(* IEC 61131-3 sources: Conveyor/test/Mocks, 7 files *)

(* ---- MockingAutoRelease copy.st ---- *)
USING Simatic.Ax.IO.Input;
NAMESPACE Simatic.Ax.Conveyor.Mocks

    CLASS MockBinSignal
        IMPLEMENTS IBinSignal
        VAR PUBLIC
            QValue : BOOL;
            QRisValue : BOOL;
            QFalValue : BOOL;
        END_VAR

        METHOD PUBLIC Q : BOOL
            Q := QValue;
        END_METHOD

        METHOD PUBLIC QRis : BOOL
            QRis := QRisValue;
        END_METHOD

        METHOD PUBLIC QFal : BOOL
            QFal := QFalValue;
        END_METHOD

        METHOD PUBLIC QBad : BOOL
            ;
        END_METHOD
END_CLASS
END_NAMESPACE

(* ---- MockingAutoRelease.st ---- *)
USING Simatic.Ax.AutomationBase;
NAMESPACE Simatic.Ax.Conveyor.Mocks

    CLASS MockAutoStartup
        IMPLEMENTS IAutoStartup
        VAR PUBLIC
            startupStatus : StartUpStatus;
        END_VAR
        METHOD PUBLIC Status : StartUpStatus
            Status := startupStatus;
        END_METHOD
    END_CLASS
END_NAMESPACE

(* ---- MockingConveyor.st ---- *)
NAMESPACE Simatic.Ax.Conveyor.Mocks

    CLASS MockingConveyor
        IMPLEMENTS IConveyor
        VAR PUBLIC
            RTD : DeliverState;
            RTR : ReceiveState;
            TIP : BOOL;
            OCC : BOOL;
        END_VAR

        METHOD PUBLIC TriggerStartInAutomatic
            ;
        END_METHOD

        METHOD PUBLIC StartManual : BOOL
            ;
        END_METHOD

        METHOD PUBLIC Stop
            ;
        END_METHOD

        METHOD PUBLIC IsOccupied : BOOL
            IsOccupied := OCC;
        END_METHOD

        METHOD PUBLIC MotorOnIsReleased : BOOL
            ;
        END_METHOD

        METHOD PUBLIC ReceiveStatus : ReceiveState
            ReceiveStatus := RTR;
        END_METHOD

        METHOD PUBLIC DeliverStatus : DeliverState
            DeliverStatus := RTD;
        END_METHOD

        METHOD PUBLIC Delivering : BOOL
            Delivering := TIP;
        END_METHOD

    METHOD PUBLIC StopSensorStatus : BOOL
        ;
    END_METHOD
END_CLASS

END_NAMESPACE

(* ---- MockingEquipment.st ---- *)
USING Simatic.Ax.AutomationBase;
NAMESPACE Simatic.Ax.Conveyor.Mocks

    CLASS MockEquiment
        IMPLEMENTS IEquipmentBase
        VAR PUBLIC
            MockError : BOOL;
            MockStatus : StartUpStatus;
            MockErrorCode : WORD;
            MockErrorText : STRING[30];
        END_VAR
        VAR PROTECTED
            _error : BOOL;
        END_VAR

        METHOD PUBLIC HasError : BOOL
            HasError := MockError;
        END_METHOD

        METHOD PUBLIC GetStartupStatus : StartUpStatus
            GetStartupStatus := MockStatus;
        END_METHOD

        METHOD PUBLIC GetError : WORD
            GetError := MockErrorCode;
        END_METHOD

        METHOD PUBLIC RunCyclic
            ;
        END_METHOD

        METHOD PUBLIC SetError
            VAR_INPUT
                errorState : WORD;
            END_VAR
            _error := TRUE;
            MockErrorCode := errorState;
        END_METHOD

        METHOD PUBLIC SetError
            VAR_INPUT
                errorState : WORD;
                errorText : STRING[30];
            END_VAR
            _error := TRUE;
            MockErrorCode := errorState;
            MockErrorText := errorText;
        END_METHOD

        METHOD PUBLIC GetErrorText : STRING[30]
            GetErrorText := MockErrorText;
        END_METHOD

        METHOD PUBLIC ResetFault
            _error := FALSE;
            MockError := FALSE;
            MockErrorCode := WORD#0;
            MockErrorText := '';
        END_METHOD
    END_CLASS

END_NAMESPACE

(* ---- MockingResetManager.st ---- *)
USING Simatic.Ax.AutomationBase;

NAMESPACE Simatic.Ax.Conveyor.Mocks

    /// Mock implementation of IResetCommand for testing
    /// Simulates reset manager behavior without actual reset logic
    CLASS MockResetManager
        IMPLEMENTS IResetCommand
        VAR PUBLIC
            /// Tracks if GetResetCommand was called
            GetResetCommandCallCount : INT := 0;
            /// Tracks if ReportError was called
            ReportErrorCallCount : INT := 0;
            /// Simulated reset command state
            ResetCommandActive : BOOL := FALSE;
        END_VAR

        /// Returns TRUE when a reset command is active
        METHOD PUBLIC ResetFaultRequest : BOOL
            GetResetCommandCallCount := GetResetCommandCallCount + 1;
            ResetFaultRequest := ResetCommandActive;
        END_METHOD

        /// Equipment calls this to report it has an active error
        METHOD PUBLIC ReportError
            ReportErrorCallCount := ReportErrorCallCount + 1;
        END_METHOD

        /// Resets the mock state for test isolation
        METHOD PUBLIC Reset
            GetResetCommandCallCount := 0;
            ReportErrorCallCount := 0;
            ResetCommandActive := FALSE;
        END_METHOD
    END_CLASS

END_NAMESPACE

(* ---- MockingStopPos.st ---- *)
NAMESPACE Simatic.Ax.Conveyor.Mocks

    CLASS MockingStopPos
        IMPLEMENTS IStopPos
        VAR PUBLIC
            Occupied : BOOL;
            Sensor : BOOL;
        END_VAR

    METHOD PUBLIC IsOccupied : BOOL
        IsOccupied := Occupied;
    END_METHOD

    METHOD PUBLIC StopSensorStatus : BOOL
        StopSensorStatus := Sensor;
    END_METHOD
END_CLASS

END_NAMESPACE

(* ---- MockMotor.st ---- *)
USING Simatic.Ax.Motor;
USING Simatic.Ax.AutomationBase;

NAMESPACE MotorTests.Mocks
    /// Mock motor for testing conveyor integration
    /// Simulates motor behavior without actual motor control
    CLASS MockMotor IMPLEMENTS IMotor
        VAR PUBLIC
            // Motor configuration properties (same as MotorGeneric)
            FixedAcceleration : LREAL := 2.0;  // m/s²
            FixedDeceleration : LREAL := 2.0;  // m/s²
            TargetSpeed : LREAL := 10.0;       // m/s
            EnableRampControl : BOOL := TRUE;

            // Test control flags
            SimulateStartFailure : BOOL := FALSE;
            SimulateAtSpeed : BOOL := TRUE;

            // Counters for test verification
            StartMotorCallCount : INT := 0;
            StopMotorCallCount : INT := 0;
        END_VAR

        VAR PROTECTED
            _isRunning : BOOL := FALSE;
            _currentSpeed : LREAL := 0.0;
            _isAtSpeed : BOOL := FALSE;
            _isReleased : BOOL := TRUE;
            _externalRelease : IRelease;
        END_VAR

        /// Starts the motor with specified parameters
        METHOD PUBLIC StartMotor
            VAR_INPUT
                targetSpeed : LREAL;
                acceleration : LREAL;
            END_VAR

            StartMotorCallCount := StartMotorCallCount + 1;

            // Update parameters if provided
            IF targetSpeed > 0.0 THEN
                THIS.TargetSpeed := targetSpeed;
            END_IF;
            IF acceleration > 0.0 THEN
                THIS.FixedAcceleration := acceleration;
            END_IF;

            IF NOT SimulateStartFailure THEN
                _isRunning := TRUE;

                // Simulate immediate speed if configured or ramp control disabled
                IF SimulateAtSpeed OR NOT EnableRampControl THEN
                    _currentSpeed := THIS.TargetSpeed;
                    _isAtSpeed := TRUE;
                ELSE
                    _currentSpeed := 0.0;
                    _isAtSpeed := FALSE;
                END_IF;
            END_IF;
        END_METHOD

        /// Stops the motor with specified deceleration
        METHOD PUBLIC StopMotor
            VAR_INPUT
                deceleration : LREAL;
            END_VAR

            StopMotorCallCount := StopMotorCallCount + 1;

            // Update deceleration if provided
            IF deceleration > 0.0 THEN
                FixedDeceleration := deceleration;
            END_IF;

            _isRunning := FALSE;
            _currentSpeed := 0.0;
            _isAtSpeed := FALSE;
        END_METHOD

        /// Returns current speed
        METHOD PUBLIC GetCurrentSpeed : LREAL
            GetCurrentSpeed := _currentSpeed;
        END_METHOD

        /// Returns whether motor is running
        METHOD PUBLIC IsRunning : BOOL
            IsRunning := _isRunning;
        END_METHOD

        /// Returns whether motor is at target speed
        METHOD PUBLIC IsAtSpeed : BOOL
            IsAtSpeed := _isAtSpeed;
        END_METHOD

        /// Returns whether motor is ramping up
        /// Always returns FALSE for mock (simplified behavior)
        METHOD PUBLIC IsRampingUp : BOOL
            IsRampingUp := FALSE;
        END_METHOD

        /// Sets the release status of the motor
        METHOD PUBLIC SetReleased
            VAR_INPUT
                released : BOOL;
            END_VAR
            _isReleased := released;
        END_METHOD

        /// Returns whether the motor is released
        METHOD PUBLIC IsReleased : BOOL
            IF _externalRelease <> NULL THEN
                IsReleased := _externalRelease.IsReleased();
            ELSE
                IsReleased := _isReleased;
            END_IF;
        END_METHOD

        /// Cyclic update method - mock implementation (does nothing)
        METHOD PUBLIC Update
            ; // Mock implementation - no operation needed
        END_METHOD

        /// Resets all counters and states
        METHOD PUBLIC Reset
            _isRunning := FALSE;
            _currentSpeed := 0.0;
            _isAtSpeed := FALSE;
            StartMotorCallCount := 0;
            StopMotorCallCount := 0;
            SimulateStartFailure := FALSE;
            SimulateAtSpeed := TRUE;
            FixedAcceleration := 2.0;
            FixedDeceleration := 2.0;
            TargetSpeed := 10.0;
            EnableRampControl := TRUE;
        END_METHOD

        /// Simulates motor reaching target speed
        METHOD PUBLIC SimulateReachTargetSpeed
            IF _isRunning THEN
                _currentSpeed := TargetSpeed;
                _isAtSpeed := TRUE;
            END_IF;
        END_METHOD
    END_CLASS
END_NAMESPACE
